SUBAPPLICATION Uebung_039_sub_NumbAnzeig (* Spiegelabfolge V2 mit Schrittkette SUB Num *)
  (* Standard: 61499-2; Description: Copyright (c) 2024 Meisterschulen am Ostbahnhof This program and the accompanying materials are made available under the terms of the Eclipse Public License 2.0 which is available at https://www.eclipse.org/legal/epl-2.0/ SPDX-License-Identifier: EPL-2.0 *)
  (* Version 1.0, 2024-03-03, Franz Höpfinger, Meisterschulen am Ostbahnhof *)
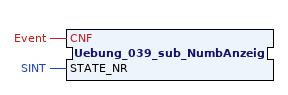
  EVENT_INPUT
    CNF;
  END_EVENT
  VAR_INPUT
    STATE_NR : SINT;
  END_VAR
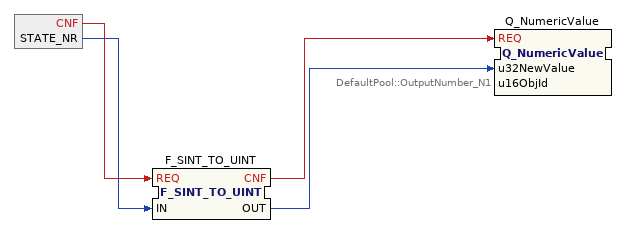
  FBS
    F_SINT_TO_UINT : F_SINT_TO_UINT;
    Q_NumericValue : Q_NumericValue(u16ObjId := DefaultPool::OutputNumber_N1);
  END_FBS
  EVENT_CONNECTIONS
    F_SINT_TO_UINT.CNF TO Q_NumericValue.REQ;
    CNF TO F_SINT_TO_UINT.REQ;
  END_CONNECTIONS
  DATA_CONNECTIONS
    F_SINT_TO_UINT.OUT TO Q_NumericValue.u32NewValue;
    STATE_NR TO F_SINT_TO_UINT.IN;
  END_CONNECTIONS
END_SUBAPPLICATION
